Fanuc KAREL source: kt00821.KL

-- PROVISIONAL review KL for V770-1; original PC SHA256 f03be5a93fd2a487b354ffa7e9d357d22de142461097a0b777e5106aab5966ba
-- Incomplete behavior may be omitted. Consult companion uncertainty JSON. Do not deploy.
PROGRAM KT00821
%NOLOCKGROUP
VAR
  I1 : INTEGER
  I2 : INTEGER
  OUT : REAL
BEGIN
  -- UNRESOLVED_PC offsets 5-16; opcodes 2E,23
  -- UNRESOLVED_PC offsets 21-32; opcodes 2E,23
  -- UNRESOLVED_PC offsets 37-48; opcodes 2E,23
  -- UNRESOLVED_PC offsets 53-64; opcodes 2E,23
  -- UNRESOLVED_PC offsets 69-86; opcodes 27,27,21,64,76,23
  -- UNRESOLVED_PC offsets 91-95; opcodes 7F
END KT00821
